{attribute 'linkalways'} 
{attribute 'no_explicit_call' := 'This FB is a CLASS and must be accessed using methods or properties'}
{attribute 'enable_dynamic_creation'}
FUNCTION_BLOCK Node_F_VN_MinElementElementwise_TcVnVector2_INT EXTENDS VisionNode
VAR
    ipContainer : _ITcVnContainer;
    aMin : _TcVnVector2_INT;
    hrPrev : _HRESULT(S_OK);
    hresult : _HRESULT(S_OK);
END_VAR

METHOD PUBLIC  Clone : I_Node
VAR
	pNode : POINTER TO Node_F_VN_MinElementElementwise_TcVnVector2_INT;
END_VAR
pNode := __NEW(Node_F_VN_MinElementElementwise_TcVnVector2_INT);
Clone := pNode^;
END_METHOD

METHOD FB_init : BOOL
VAR_INPUT
	bInitRetains : BOOL; // if TRUE, the retain variables are initialized (warm start / cold start)
	bInCopyCode : BOOL;  // if TRUE, the instance afterwards gets moved into the copy code (online change)
END_VAR
AddInput('ipContainer', ipContainer);
AddInput('hrPrev', hrPrev);
AddOutput('ipContainer', ipContainer);
AddOutput('aMin', aMin);
AddOutput('hresult',hresult);
END_METHOD

METHOD PROTECTED OnExecute
hresult.Value := F_VN_MinElementElementwise_TcVnVector2_INT(
    ipContainer := ipContainer.Value,
    aMin := aMin.Value,
    hrPrev:= hrPrev.Value);
END_METHOD

METHOD PUBLIC PreExecutionCheck
VAR_INPUT
	Check : I_PreExecutionChecks;
END_VAR
Check.IsTrue(ipContainer.IsValid, 'ipContainer must be a valid container');
Check.IsTrue(ipContainer.IsType(TC_GLOBAL_CONST_LIST.ContainerType_Vector_TcVnVector2_INT), 'ipContainer contains incorrect type');
END_METHOD

END_FUNCTION_BLOCK

(* stored: Version 1.1.0.1, ProductVersion 3.1.4026.13
   POU Node_F_VN_MinElementElementwise_TcVnVector2_INT: Id {9c954cb6-b723-42c2-a07c-308892f6ecf3}, SpecialFunc None
   Folder Constructor: Id {2e94b136-e0fc-4802-97cb-896d7a242ee4}
   Method Clone: Id {73792f1c-d560-4274-826c-4b49787cd20c}
   Method FB_init: Id {4cd26c2f-0fa6-4115-8943-0db74e0400ca}
   Method OnExecute: Id {6468e499-f144-4a8d-baf0-b8f38f509e8c}
   Method PreExecutionCheck: Id {9ee02b95-d538-4c8b-9c70-c2046175d088} *)
